Omron CX-Programmer project NewProject (CX-Programmer 9.50)

# PLC coba: CP1L M

## Global symbols (name address type ; comment)
0.05 BOOL  ; baterai diaktifkan discharge
10.00 BOOL  ; Battery aktif
20.00 BOOL  ; kabel 1 blok 1
20.01 BOOL  ; kabel 2 blok 1
20.02 BOOL  ; kabel 3 blok 1
20.03 BOOL  ; kabel 4 blok 1
20.04 BOOL  ; kabel 5 blok 1
20.05 BOOL  ; Kabel transmisi pv1 blok 2 dan cos 1
20.06 BOOL  ; Kabel transmisi pv2 blok 2 dan cos 2
20.07 BOOL  ; Kabel transmisi pv3 blok 2 dan cos 3
20.08 BOOL  ; Kabel transmisi pv4 blok2 dan cos4
20.09 BOOL  ; Kabel transmisi pv5 blok 2 dan cos 5
20.10 BOOL  ; kabel transmisi dan cos pada battery
20.12 BOOL  ; panah battery
25.00 BOOL  ; giliran pv2
25.01 BOOL  ; giliran pv3
25.02 BOOL  ; giliran pv4
25.03 BOOL  ; giliran pv5
A341 CHANNEL  ; hh:mm:ss
A342 CHANNEL  ; hh:mm:ss
A351 CHANNEL  ; hh:mm:ss
D0 CHANNEL  ; pv 1
D1 CHANNEL  ; pv 2
D10 CHANNEL  ; Transmisi PV 4
D101 CHANNEL  ; jam aktif
D11 CHANNEL  ; Transmisi PV 5
D111 CHANNEL  ; jam mati
D12 CHANNEL  ; Transmisi atau Receive Battery
D2 CHANNEL  ; pv 3
D20 CHANNEL  ; Be-B1
D21 CHANNEL  ; D20 - B2
D22 CHANNEL  ; D21 - B3
D23 CHANNEL  ; D22 - B4
D24 CHANNEL  ; D23 - B5
D3 CHANNEL  ; pv 4
D4 CHANNEL  ; pv5
D5 CHANNEL  ; Kondisi battery
D6 CHANNEL  ; Kebutuhan beban
D7 CHANNEL  ; Transmisi PV 1
D70 CHANNEL  ; jumlah pv1 + pv2
D71 CHANNEL  ; jumlah pv3 + pv4
D72 CHANNEL  ; jumlah pv 1 sd 4
D73 CHANNEL  ; jumlah pv 1 sd 5
D74 CHANNEL  ; tTransmisi PV 1 & 2
D75 CHANNEL  ; Transmisi PV 3 & 4
D76 CHANNEL  ; Transmisi PV 1 sd 4
D77 CHANNEL  ; Transmisi PV 1 sd  5
D8 CHANNEL  ; Transmisi PV 2
D80 CHANNEL  ; selisih full - kapasitas sekarang
D81 CHANNEL  ; d80 bagi d12
D82 CHANNEL  ; pengisian daya perdetik
D9 CHANNEL  ; Transmisi PV 3
W0.00 BOOL  ; START
W0.01 BOOL  ; Battery aktif karena di luar jam kerja pv

## Program NewProgram1 (cyclic task 0)
Local symbols
F110 REAL

### Section Section1

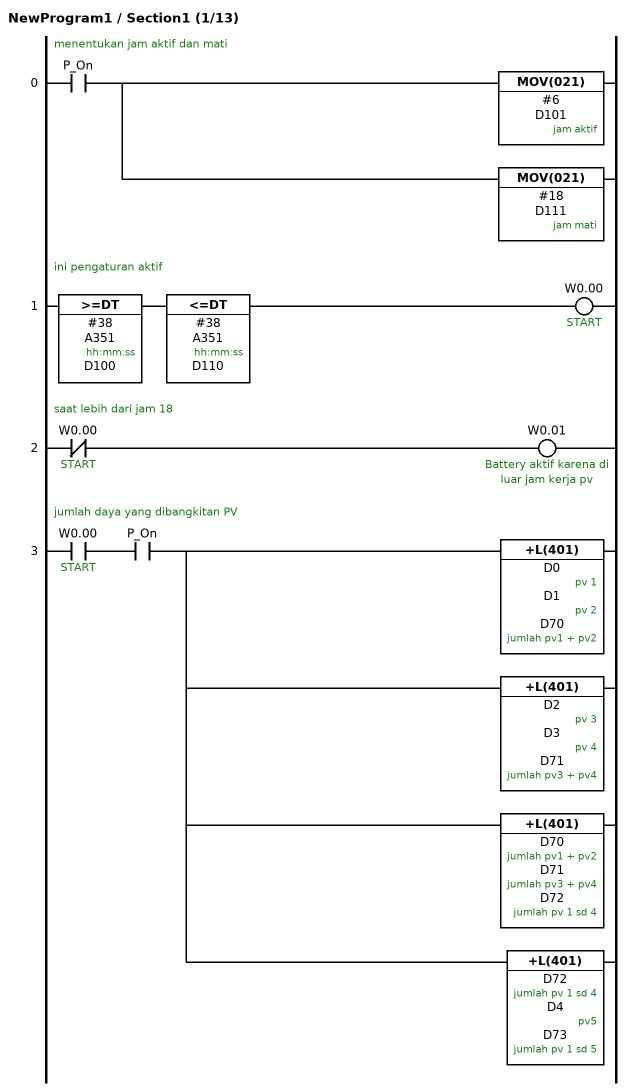
; rung 0: menentukan jam aktif dan mati
LD P_On
MOV(021) #6 D101  ; jam aktif
MOV(021) #18 D111  ; jam mati
; rung 1: ini pengaturan aktif
LD>=DT(346) #38 A351 D100  ; hh:mm:ss
AND<=DT(344) #38 A351 D110  ; hh:mm:ss
OUT W0.00  ; START
; rung 2: saat lebih dari jam 18
LDNOT W0.00  ; START
OUT W0.01  ; Battery aktif karena di luar jam kerja pv
; rung 3: jumlah daya yang dibangkitan PV
LD W0.00  ; START
AND P_On
+L(401) D0 D1 D70  ; pv 1, pv 2, jumlah pv1 + pv2
+L(401) D2 D3 D71  ; pv 3, pv 4, jumlah pv3 + pv4
+L(401) D70 D71 D72  ; jumlah pv1 + pv2, jumlah pv3 + pv4, jumlah pv 1 sd 4
+L(401) D72 D4 D73  ; jumlah pv 1 sd 4, pv5, jumlah pv 1 sd 5

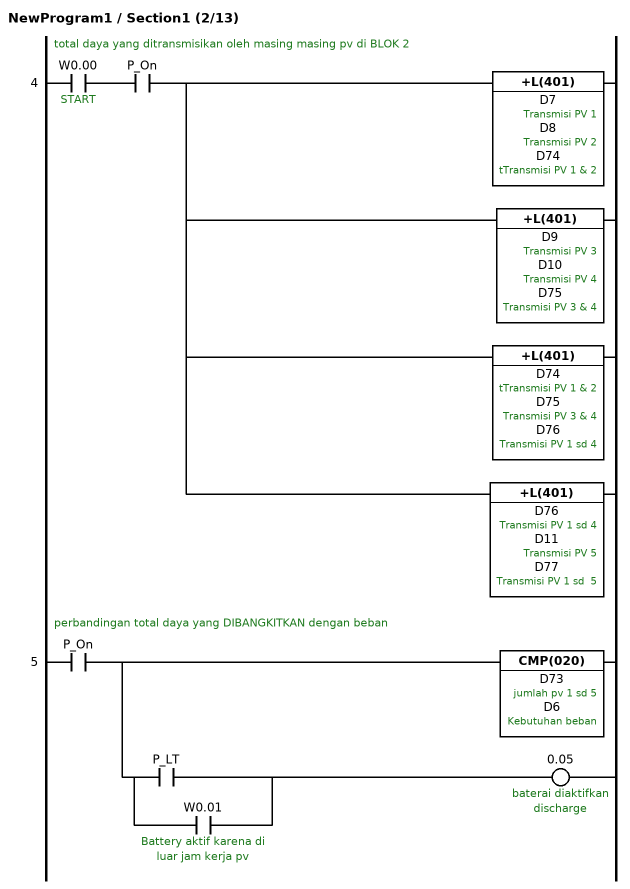
; rung 4: total daya yang ditransmisikan oleh masing masing pv di BLOK 2
LD W0.00  ; START
AND P_On
+L(401) D7 D8 D74  ; Transmisi PV 1, Transmisi PV 2, tTransmisi PV 1 & 2
+L(401) D9 D10 D75  ; Transmisi PV 3, Transmisi PV 4, Transmisi PV 3 & 4
+L(401) D74 D75 D76  ; tTransmisi PV 1 & 2, Transmisi PV 3 & 4, Transmisi PV 1 sd 4
+L(401) D76 D11 D77  ; Transmisi PV 1 sd 4, Transmisi PV 5, Transmisi PV 1 sd  5
; rung 5: perbandingan total daya yang DIBANGKITKAN dengan beban
LD P_On
CMP(020) D73 D6  ; jumlah pv 1 sd 5, Kebutuhan beban
LD P_LT
OR W0.01  ; Battery aktif karena di luar jam kerja pv
ANDLD
OUT 0.05  ; baterai diaktifkan discharge

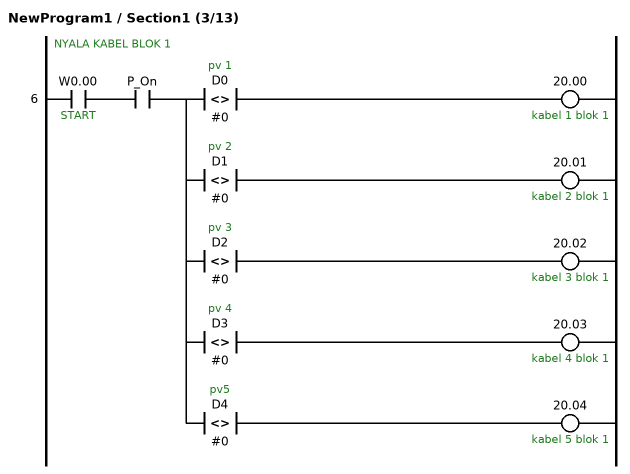
; rung 6: NYALA KABEL BLOK 1
LD W0.00  ; START
AND P_On
OUT TR0
AND<>(305) D0 #0  ; pv 1
OUT 20.00  ; kabel 1 blok 1
LD TR0
AND<>(305) D1 #0  ; pv 2
OUT 20.01  ; kabel 2 blok 1
LD TR0
AND<>(305) D2 #0  ; pv 3
OUT 20.02  ; kabel 3 blok 1
LD TR0
AND<>(305) D3 #0  ; pv 4
OUT 20.03  ; kabel 4 blok 1
LD TR0
AND<>(305) D4 #0  ; pv5
OUT 20.04  ; kabel 5 blok 1

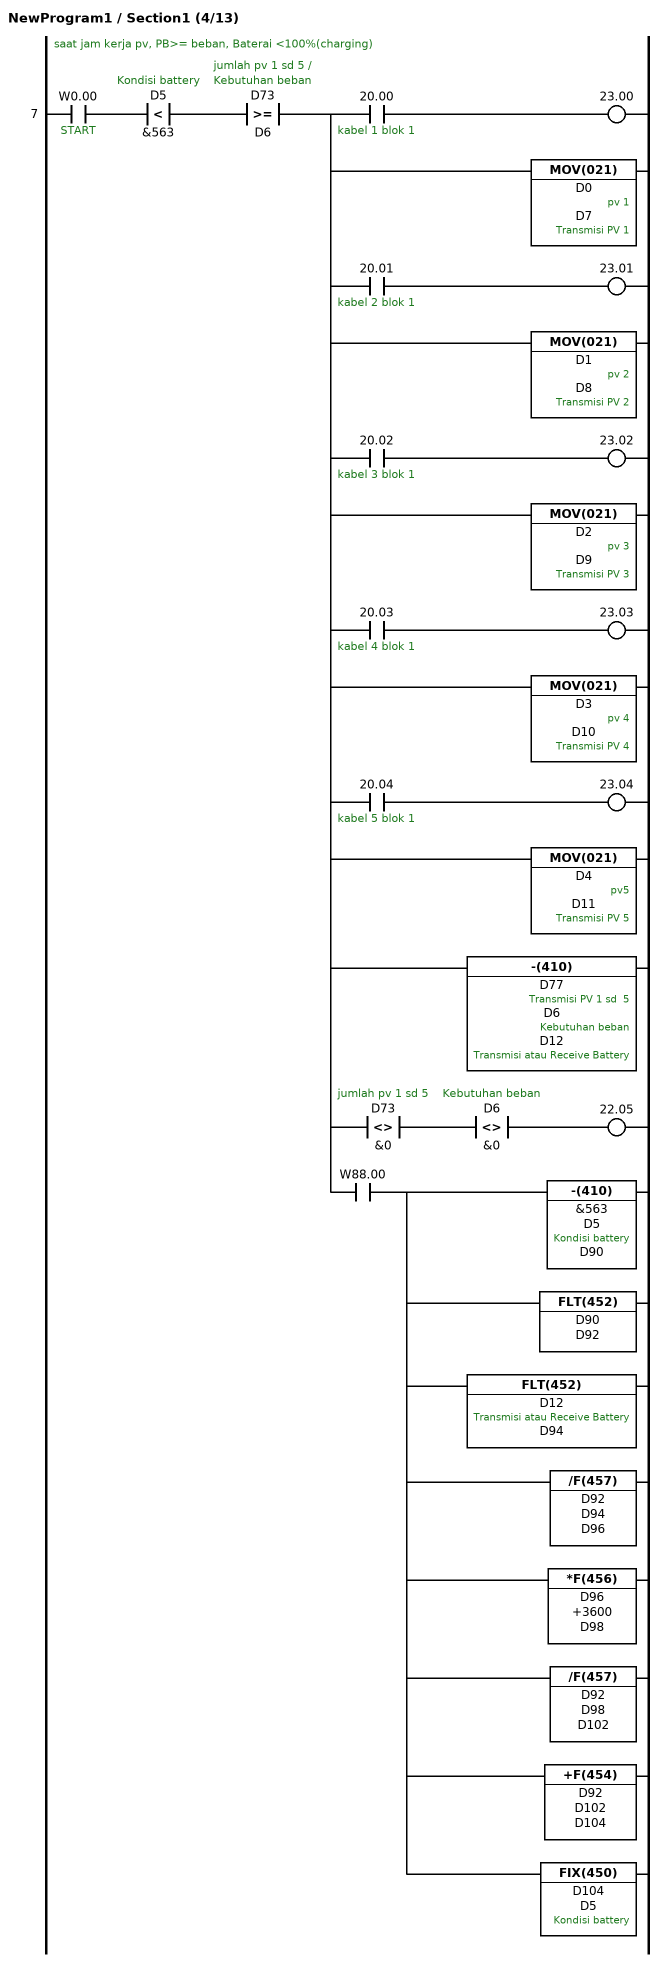
; rung 7: saat jam kerja pv, PB>= beban, Baterai <100%(charging)
LD W0.00  ; START
AND<(310) D5 &563  ; Kondisi battery
AND>=(325) D73 D6  ; jumlah pv 1 sd 5, Kebutuhan beban
OUT TR0
AND 20.00  ; kabel 1 blok 1
OUT 23.00
LD TR0
MOV(021) D0 D7  ; pv 1, Transmisi PV 1
AND 20.01  ; kabel 2 blok 1
OUT 23.01
LD TR0
MOV(021) D1 D8  ; pv 2, Transmisi PV 2
AND 20.02  ; kabel 3 blok 1
OUT 23.02
LD TR0
MOV(021) D2 D9  ; pv 3, Transmisi PV 3
AND 20.03  ; kabel 4 blok 1
OUT 23.03
LD TR0
MOV(021) D3 D10  ; pv 4, Transmisi PV 4
AND 20.04  ; kabel 5 blok 1
OUT 23.04
LD TR0
MOV(021) D4 D11  ; pv5, Transmisi PV 5
-(410) D77 D6 D12  ; Transmisi PV 1 sd  5, Kebutuhan beban, Transmisi atau Receive Battery
AND<>S(307) D73 &0  ; jumlah pv 1 sd 5
AND<>S(307) D6 &0  ; Kebutuhan beban
OUT 22.05
LD TR0
AND W88.00
-(410) &563 D5 D90  ; Kondisi battery
FLT(452) D90 D92
FLT(452) D12 D94  ; Transmisi atau Receive Battery
/F(457) D92 D94 D96
*F(456) D96 +3600 D98
/F(457) D92 D98 D102
+F(454) D92 D102 D104
FIX(450) D104 D5  ; Kondisi battery

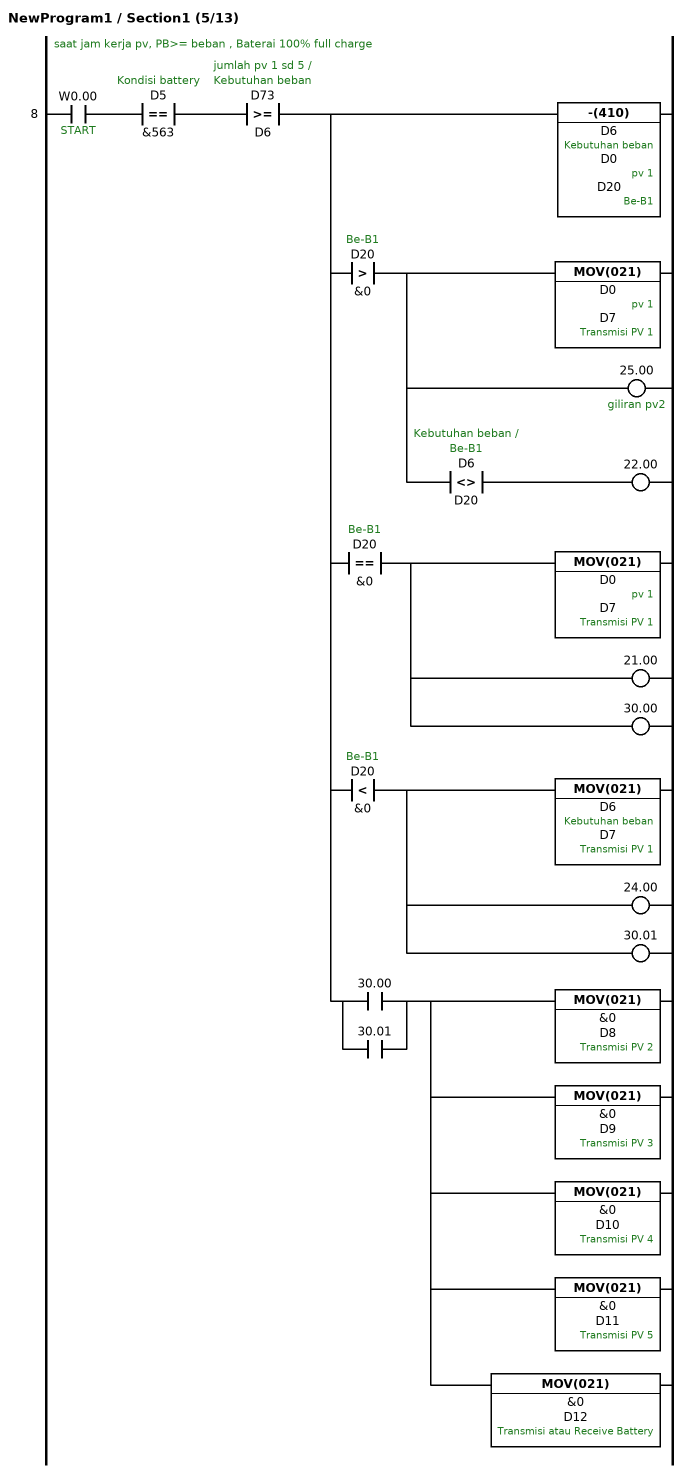
; rung 8: saat jam kerja pv, PB>= beban , Baterai 100% full charge
LD W0.00  ; START
AND=(300) D5 &563  ; Kondisi battery
AND>=(325) D73 D6  ; jumlah pv 1 sd 5, Kebutuhan beban
OUT TR0
-(410) D6 D0 D20  ; Kebutuhan beban, pv 1, Be-B1
AND>S(322) D20 &0  ; Be-B1
MOV(021) D0 D7  ; pv 1, Transmisi PV 1
OUT 25.00  ; giliran pv2
AND<>S(307) D6 D20  ; Kebutuhan beban, Be-B1
OUT 22.00
LD TR0
AND=S(302) D20 &0  ; Be-B1
MOV(021) D0 D7  ; pv 1, Transmisi PV 1
OUT 21.00
OUT 30.00
LD TR0
AND<S(312) D20 &0  ; Be-B1
MOV(021) D6 D7  ; Kebutuhan beban, Transmisi PV 1
OUT 24.00
OUT 30.01
LD TR0
LD 30.00
OR 30.01
ANDLD
MOV(021) &0 D8  ; Transmisi PV 2
MOV(021) &0 D9  ; Transmisi PV 3
MOV(021) &0 D10  ; Transmisi PV 4
MOV(021) &0 D11  ; Transmisi PV 5
MOV(021) &0 D12  ; Transmisi atau Receive Battery

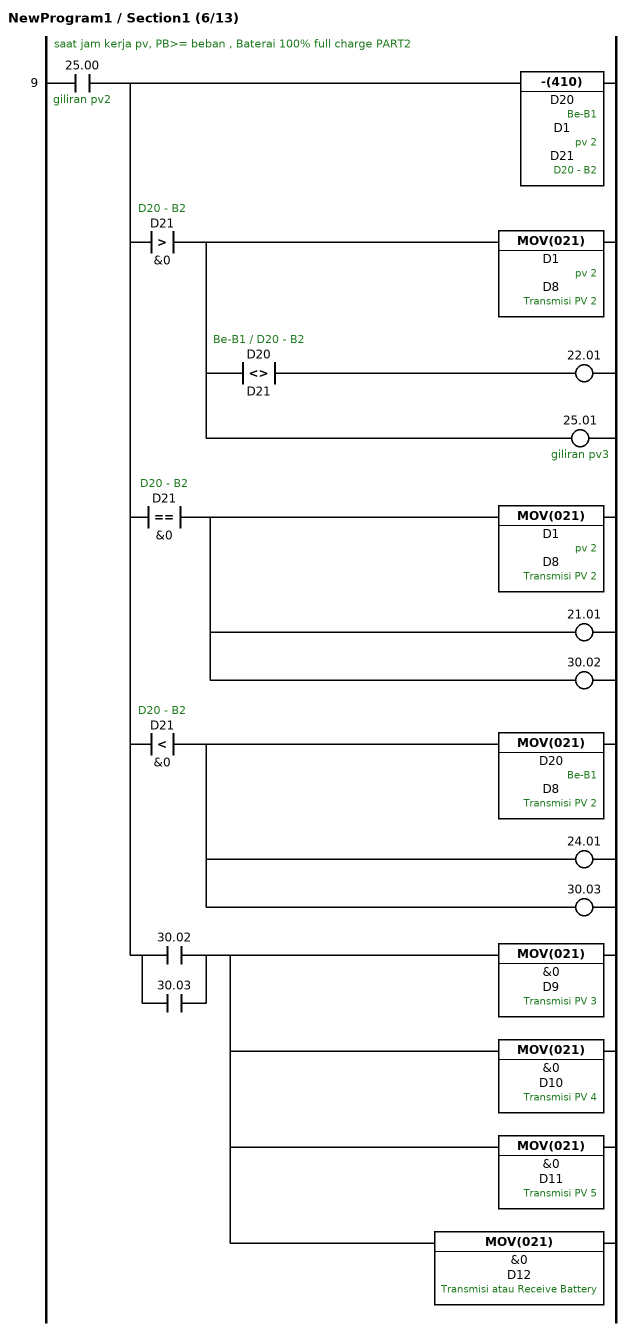
; rung 9: saat jam kerja pv, PB>= beban , Baterai 100% full charge PART2
LD 25.00  ; giliran pv2
OUT TR0
-(410) D20 D1 D21  ; Be-B1, pv 2, D20 - B2
AND>S(322) D21 &0  ; D20 - B2
OUT TR1
MOV(021) D1 D8  ; pv 2, Transmisi PV 2
AND<>S(307) D20 D21  ; Be-B1, D20 - B2
OUT 22.01
LD TR1
OUT 25.01  ; giliran pv3
LD TR0
AND=S(302) D21 &0  ; D20 - B2
MOV(021) D1 D8  ; pv 2, Transmisi PV 2
OUT 21.01
OUT 30.02
LD TR0
AND<S(312) D21 &0  ; D20 - B2
MOV(021) D20 D8  ; Be-B1, Transmisi PV 2
OUT 24.01
OUT 30.03
LD TR0
LD 30.02
OR 30.03
ANDLD
MOV(021) &0 D9  ; Transmisi PV 3
MOV(021) &0 D10  ; Transmisi PV 4
MOV(021) &0 D11  ; Transmisi PV 5
MOV(021) &0 D12  ; Transmisi atau Receive Battery

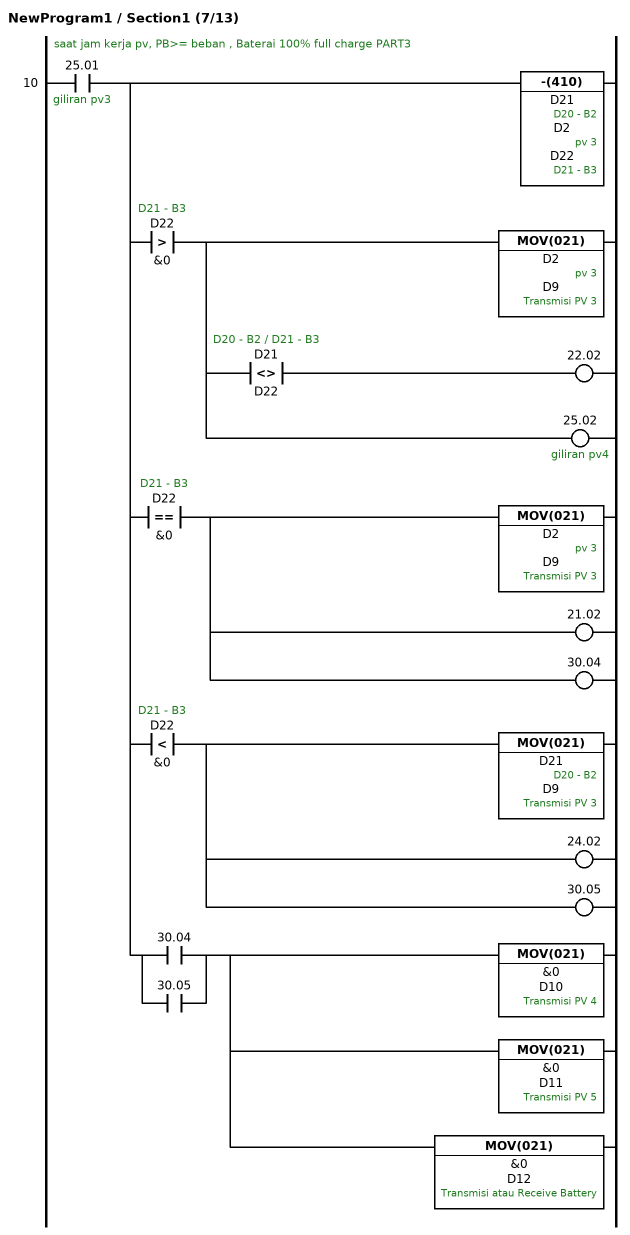
; rung 10: saat jam kerja pv, PB>= beban , Baterai 100% full charge PART3
LD 25.01  ; giliran pv3
OUT TR0
-(410) D21 D2 D22  ; D20 - B2, pv 3, D21 - B3
AND>S(322) D22 &0  ; D21 - B3
OUT TR1
MOV(021) D2 D9  ; pv 3, Transmisi PV 3
AND<>S(307) D21 D22  ; D20 - B2, D21 - B3
OUT 22.02
LD TR1
OUT 25.02  ; giliran pv4
LD TR0
AND=S(302) D22 &0  ; D21 - B3
MOV(021) D2 D9  ; pv 3, Transmisi PV 3
OUT 21.02
OUT 30.04
LD TR0
AND<S(312) D22 &0  ; D21 - B3
MOV(021) D21 D9  ; D20 - B2, Transmisi PV 3
OUT 24.02
OUT 30.05
LD TR0
LD 30.04
OR 30.05
ANDLD
MOV(021) &0 D10  ; Transmisi PV 4
MOV(021) &0 D11  ; Transmisi PV 5
MOV(021) &0 D12  ; Transmisi atau Receive Battery

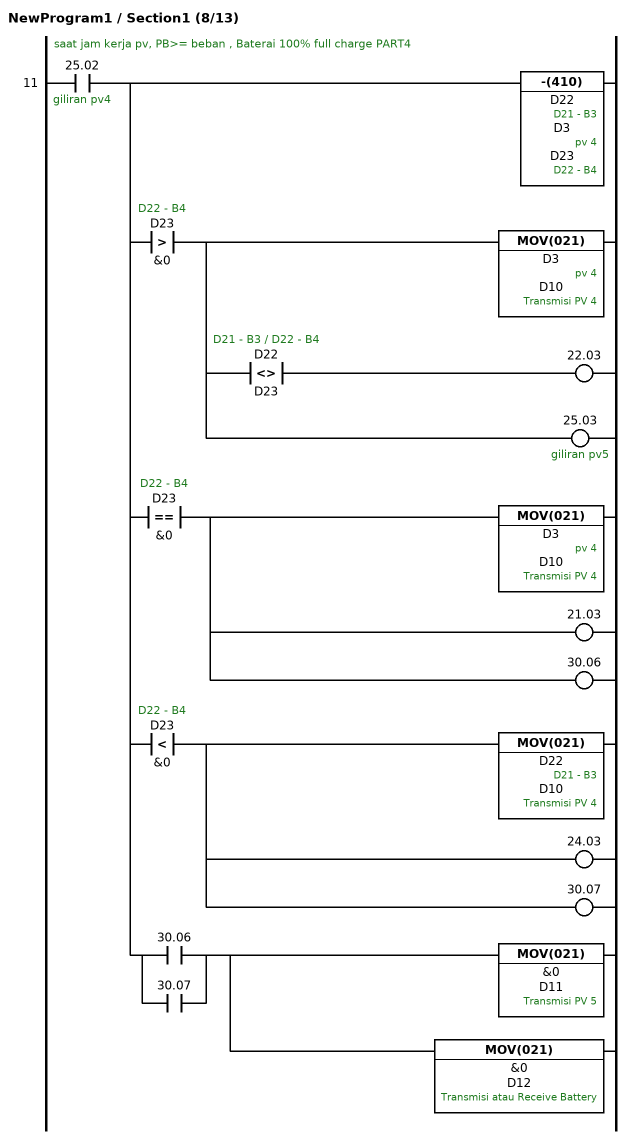
; rung 11: saat jam kerja pv, PB>= beban , Baterai 100% full charge PART4
LD 25.02  ; giliran pv4
OUT TR0
-(410) D22 D3 D23  ; D21 - B3, pv 4, D22 - B4
AND>S(322) D23 &0  ; D22 - B4
OUT TR1
MOV(021) D3 D10  ; pv 4, Transmisi PV 4
AND<>S(307) D22 D23  ; D21 - B3, D22 - B4
OUT 22.03
LD TR1
OUT 25.03  ; giliran pv5
LD TR0
AND=S(302) D23 &0  ; D22 - B4
MOV(021) D3 D10  ; pv 4, Transmisi PV 4
OUT 21.03
OUT 30.06
LD TR0
AND<S(312) D23 &0  ; D22 - B4
MOV(021) D22 D10  ; D21 - B3, Transmisi PV 4
OUT 24.03
OUT 30.07
LD TR0
LD 30.06
OR 30.07
ANDLD
MOV(021) &0 D11  ; Transmisi PV 5
MOV(021) &0 D12  ; Transmisi atau Receive Battery

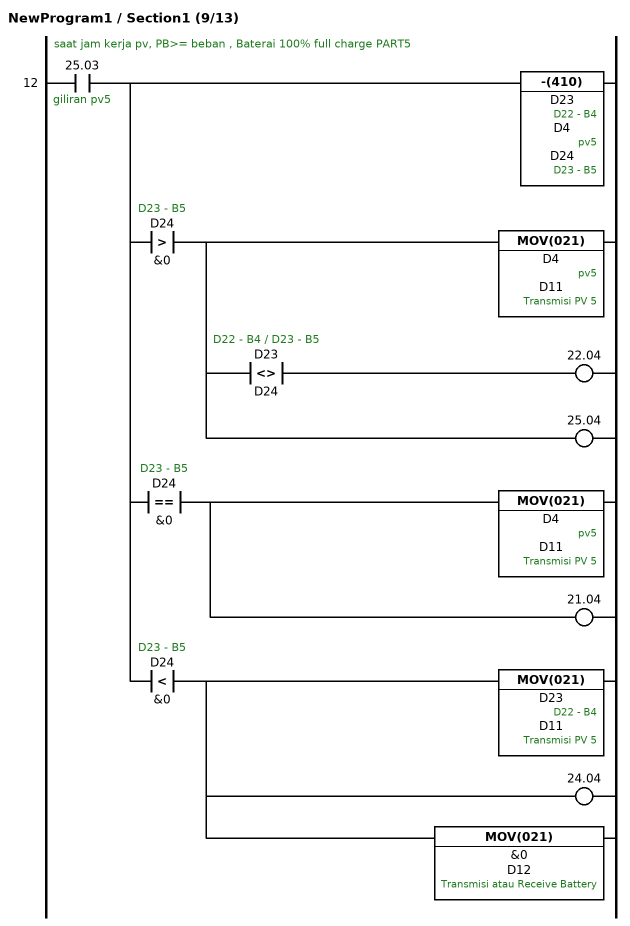
; rung 12: saat jam kerja pv, PB>= beban , Baterai 100% full charge PART5
LD 25.03  ; giliran pv5
OUT TR0
-(410) D23 D4 D24  ; D22 - B4, pv5, D23 - B5
AND>S(322) D24 &0  ; D23 - B5
OUT TR1
MOV(021) D4 D11  ; pv5, Transmisi PV 5
AND<>S(307) D23 D24  ; D22 - B4, D23 - B5
OUT 22.04
LD TR1
OUT 25.04
LD TR0
AND=S(302) D24 &0  ; D23 - B5
MOV(021) D4 D11  ; pv5, Transmisi PV 5
OUT 21.04
LD TR0
AND<S(312) D24 &0  ; D23 - B5
MOV(021) D23 D11  ; D22 - B4, Transmisi PV 5
OUT 24.04
MOV(021) &0 D12  ; Transmisi atau Receive Battery

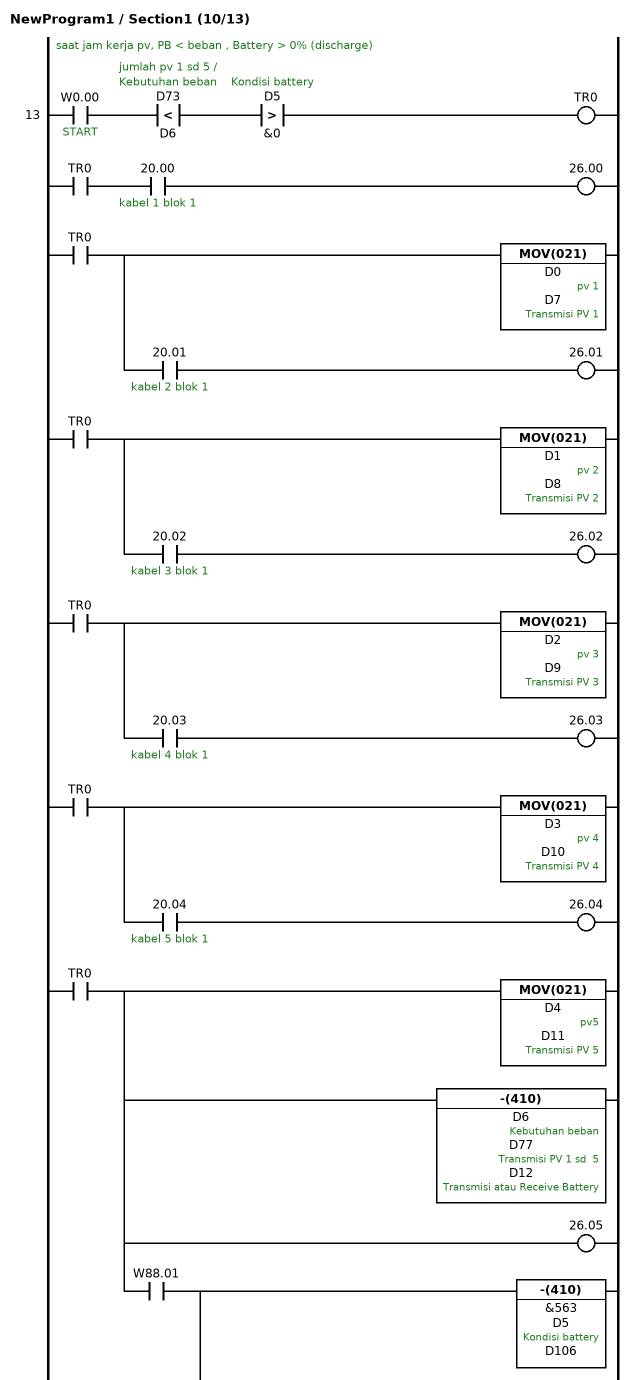

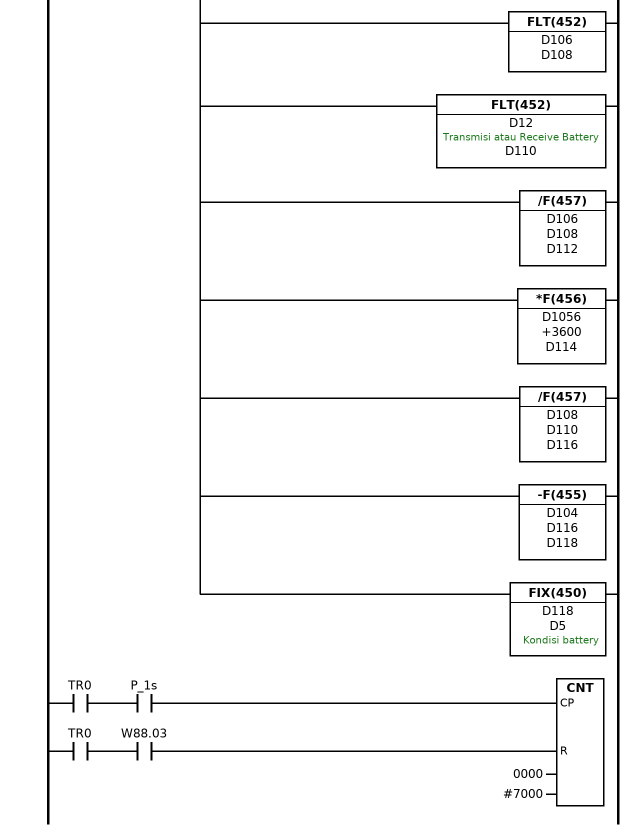
; rung 13: saat jam kerja pv, PB < beban , Battery > 0% (discharge)
LD W0.00  ; START
AND<S(312) D73 D6  ; jumlah pv 1 sd 5, Kebutuhan beban
AND>S(322) D5 &0  ; Kondisi battery
OUT TR0
AND 20.00  ; kabel 1 blok 1
OUT 26.00
LD TR0
MOV(021) D0 D7  ; pv 1, Transmisi PV 1
AND 20.01  ; kabel 2 blok 1
OUT 26.01
LD TR0
MOV(021) D1 D8  ; pv 2, Transmisi PV 2
AND 20.02  ; kabel 3 blok 1
OUT 26.02
LD TR0
MOV(021) D2 D9  ; pv 3, Transmisi PV 3
AND 20.03  ; kabel 4 blok 1
OUT 26.03
LD TR0
MOV(021) D3 D10  ; pv 4, Transmisi PV 4
AND 20.04  ; kabel 5 blok 1
OUT 26.04
LD TR0
MOV(021) D4 D11  ; pv5, Transmisi PV 5
-(410) D6 D77 D12  ; Kebutuhan beban, Transmisi PV 1 sd  5, Transmisi atau Receive Battery
OUT 26.05
AND W88.01
-(410) &563 D5 D106  ; Kondisi battery
FLT(452) D106 D108
FLT(452) D12 D110  ; Transmisi atau Receive Battery
/F(457) D106 D108 D112
*F(456) D1056 +3600 D114
/F(457) D108 D110 D116
-F(455) D104 D116 D118
FIX(450) D118 D5  ; Kondisi battery
LD TR0
AND P_1s
LD TR0
AND W88.03
CNT 0000 #7000
; rung 14: saat jam kerja pv, PB < beban, battery 0%

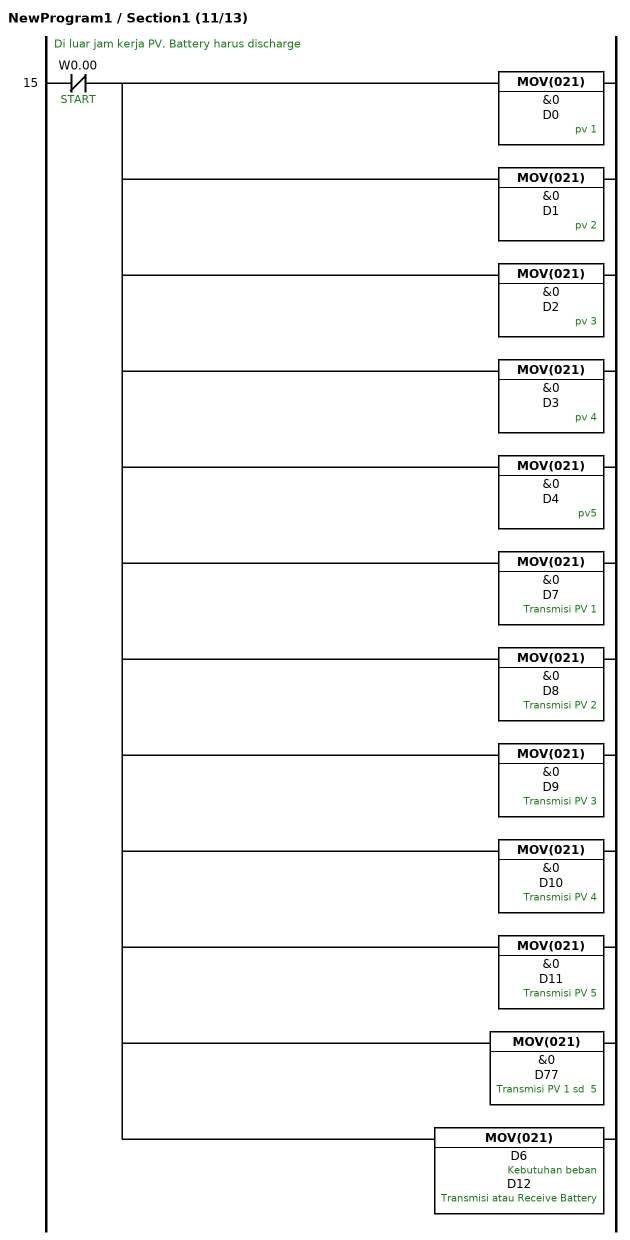
; rung 15: Di luar jam kerja PV. Battery harus discharge
LDNOT W0.00  ; START
MOV(021) &0 D0  ; pv 1
MOV(021) &0 D1  ; pv 2
MOV(021) &0 D2  ; pv 3
MOV(021) &0 D3  ; pv 4
MOV(021) &0 D4  ; pv5
MOV(021) &0 D7  ; Transmisi PV 1
MOV(021) &0 D8  ; Transmisi PV 2
MOV(021) &0 D9  ; Transmisi PV 3
MOV(021) &0 D10  ; Transmisi PV 4
MOV(021) &0 D11  ; Transmisi PV 5
MOV(021) &0 D77  ; Transmisi PV 1 sd  5
MOV(021) D6 D12  ; Kebutuhan beban, Transmisi atau Receive Battery

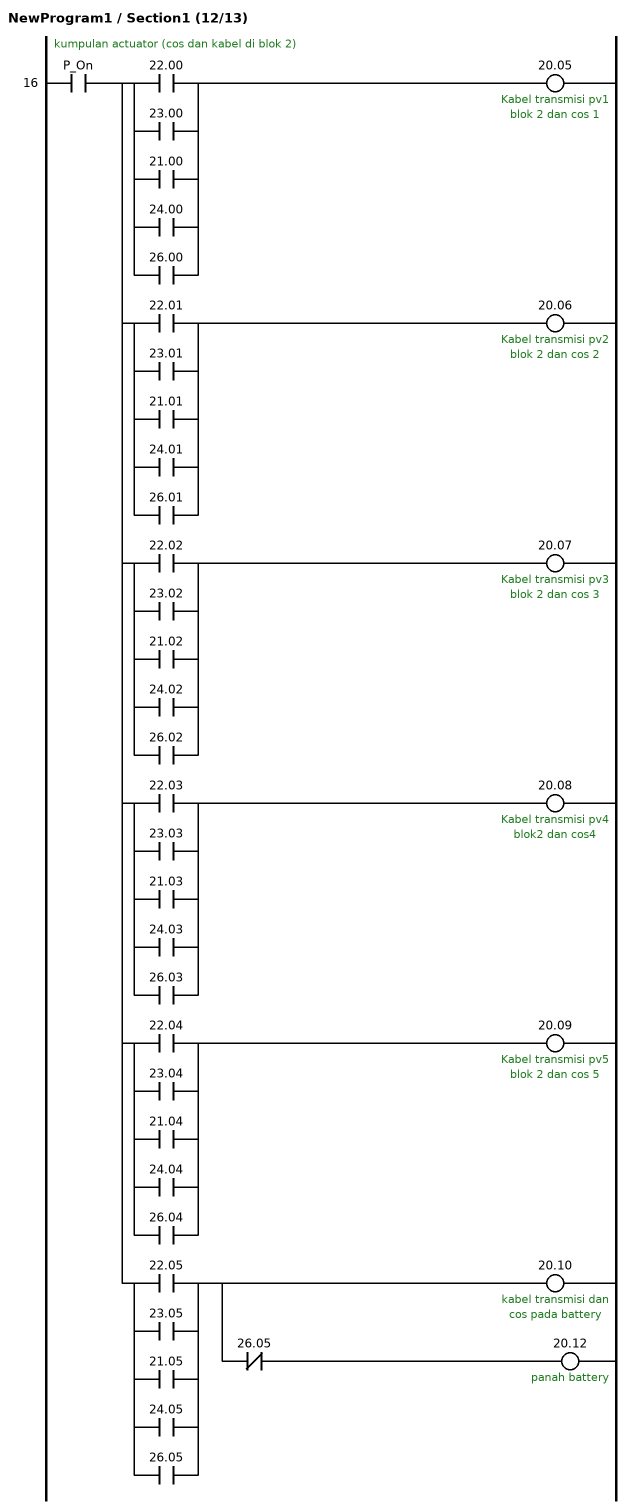
; rung 16: kumpulan actuator (cos dan kabel di blok 2)
LD P_On
OUT TR0
LD 22.00
OR 23.00
OR 21.00
OR 24.00
OR 26.00
ANDLD
OUT 20.05  ; Kabel transmisi pv1 blok 2 dan cos 1
LD TR0
LD 22.01
OR 23.01
OR 21.01
OR 24.01
OR 26.01
ANDLD
OUT 20.06  ; Kabel transmisi pv2 blok 2 dan cos 2
LD TR0
LD 22.02
OR 23.02
OR 21.02
OR 24.02
OR 26.02
ANDLD
OUT 20.07  ; Kabel transmisi pv3 blok 2 dan cos 3
LD TR0
LD 22.03
OR 23.03
OR 21.03
OR 24.03
OR 26.03
ANDLD
OUT 20.08  ; Kabel transmisi pv4 blok2 dan cos4
LD TR0
LD 22.04
OR 23.04
OR 21.04
OR 24.04
OR 26.04
ANDLD
OUT 20.09  ; Kabel transmisi pv5 blok 2 dan cos 5
LD TR0
LD 22.05
OR 23.05
OR 21.05
OR 24.05
OR 26.05
ANDLD
OUT 20.10  ; kabel transmisi dan cos pada battery
ANDNOT 26.05
OUT 20.12  ; panah battery

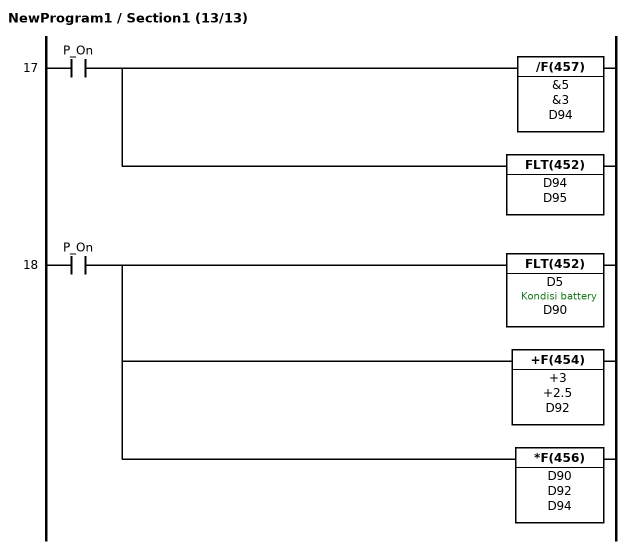
; rung 17
LD P_On
/F(457) &5 &3 D94
FLT(452) D94 D95
; rung 18
LD P_On
FLT(452) D5 D90  ; Kondisi battery
+F(454) +3 +2.5 D92
*F(456) D90 D92 D94

### Section END
; rung 0
END(001)